(* PLC project Sin nombre, Desconocido Sin nombre 1 *)
(* stored: creationDateTime 2025-06-17T15:10:20, modificationDateTime 2025-06-17T15:31:40 *)

PROGRAM Main
  VAR
    xApertura_Valv_Alim : BOOL;
    xArranque_Motor_Agit : BOOL;
    xApertura_Valv_Fluido : BOOL;
    xApertura_Valv_Desc : BOOL;
    xComando_Arranque : BOOL;
    xTanque_Lleno : BOOL;
    xTanque_Vacio : BOOL;
    xEtapa3 : BOOL;
    TON0 : TON;
  END_VAR

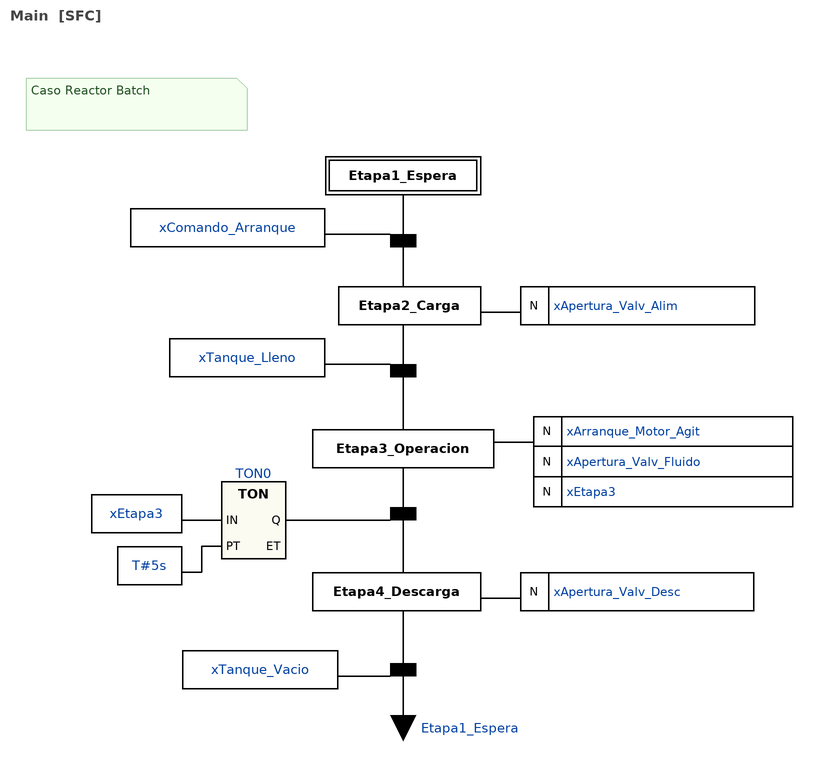
(* Caso Reactor Batch *)
INITIAL_STEP Etapa1_Espera:
  COMPUTE_FUNCTION_BLOCKS(S);
END_STEP
TRANSITION FROM Etapa1_Espera TO Etapa2_Carga
  := xComando_Arranque;
END_TRANSITION
STEP Etapa2_Carga:
  xApertura_Valv_Alim(N);
END_STEP
TRANSITION FROM Etapa2_Carga TO Etapa3_Operacion
  := xTanque_Lleno;
END_TRANSITION
STEP Etapa3_Operacion:
  xArranque_Motor_Agit(N);
  xApertura_Valv_Fluido(N);
  xEtapa3(N);
END_STEP
TRANSITION FROM Etapa3_Operacion TO Etapa4_Descarga
  := TON0.Q;
END_TRANSITION
STEP Etapa4_Descarga:
  xApertura_Valv_Desc(N);
END_STEP
TRANSITION FROM Etapa4_Descarga TO Etapa1_Espera
  := xTanque_Vacio;
END_TRANSITION
ACTION COMPUTE_FUNCTION_BLOCKS:  (* blocks drawn on the SFC sheet *)
  TON0(IN := xEtapa3, PT := T#5s);
END_ACTION
END_PROGRAM

CONFIGURATION Config0
  RESOURCE Res0 ON PLC
    TASK task0(INTERVAL := T#20ms, PRIORITY := 0);
    PROGRAM instance0 WITH task0 : Main;
  END_RESOURCE
END_CONFIGURATION
